Omron Sysmac Studio project SorterKonveyor (Sysmac Studio 1.65.0.64007, StandardProject)

# Controller new_Controller_0: NX1P2-1040DT1 version 1.69
Task PrimaryTask (priority 4, period or condition 2000): Program0

VAR_GLOBAL
    BIO_Input_Bit_00 : BOOL;  (* at BuiltInIO://cpu/#0/Input_Bit_00 *)
    BIO_Input_Bit_01 : BOOL;  (* at BuiltInIO://cpu/#0/Input_Bit_01 *)
    BIO_Input_Bit_02 : BOOL;  (* at BuiltInIO://cpu/#0/Input_Bit_02 *)
    BIO_Input_Bit_03 : BOOL;  (* at BuiltInIO://cpu/#0/Input_Bit_03 *)
    BIO_Input_Bit_04 : BOOL;  (* at BuiltInIO://cpu/#0/Input_Bit_04 *)
    BIO_Input_Bit_05 : BOOL;  (* at BuiltInIO://cpu/#0/Input_Bit_05 *)
    BIO_Input_Bit_06 : BOOL;  (* at BuiltInIO://cpu/#0/Input_Bit_06 *)
    BIO_Input_Bit_07 : BOOL;  (* at BuiltInIO://cpu/#0/Input_Bit_07 *)
    BIO_Output_Bit_00 : BOOL;  (* at BuiltInIO://cpu/#0/Output_Bit_00 *)
    BIO_Output_Bit_01 : BOOL;  (* at BuiltInIO://cpu/#0/Output_Bit_01 *)
    BIO_Output_Bit_02 : BOOL;  (* at BuiltInIO://cpu/#0/Output_Bit_02 *)
    BIO_Output_Bit_03 : BOOL;  (* at BuiltInIO://cpu/#0/Output_Bit_03 *)
    BIO_Output_Bit_04 : BOOL;  (* at BuiltInIO://cpu/#0/Output_Bit_04 *)
    BIO_Output_Bit_05 : BOOL;  (* at BuiltInIO://cpu/#0/Output_Bit_05 *)
    BIO_Output_Bit_06 : BOOL;  (* at BuiltInIO://cpu/#0/Output_Bit_06 *)
    BIO_Output_Bit_07 : BOOL;  (* at BuiltInIO://cpu/#0/Output_Bit_07 *)
    BIO_Output_Bit_08 : BOOL;  (* at BuiltInIO://cpu/#0/Output_Bit_08 *)
    BIO_Output_Bit_09 : BOOL;  (* at BuiltInIO://cpu/#0/Output_Bit_09 *)
    IN_Start_But : BOOL;
    IN_Stop_But : BOOL;
    IN_Motor0_Ariza : BOOL;
    IN_Motor1_Ariza : BOOL;
    IN_Motor3_Ariza : BOOL;
    IN_Motor2_Ariza : BOOL;
    IN_Motor4_Ariza : BOOL;
    OUT_Motor0_İleri : BOOL;
    OUT_Motor0_Geri : BOOL;
    OUT_Motor1_İleri : BOOL;
    OUT_Motor1_Geri : BOOL;
    OUT_Motor2_İleri : BOOL;
    OUT_Motor2_Geri : BOOL;
    OUT_Motor3_İleri : BOOL;
    OUT_Motor3_Geri : BOOL;
    OUT_Motor4_İleri : BOOL;
    OUT_Motor4_Geri : BOOL;
    OUT_Buzzer : BOOL;
    IN_Urun_Algilama_Sens : BOOL;
    ALARM : ARRAY[0..50] OF BOOL;
    Barcode_Info : STRING[10];
    Product_Cycle : INT;
    Barcode_Regsiter1 : STRING[10];
    Barcode_Regsiter2 : STRING[10];
    Barcode_Regsiter3 : STRING[10];
    Barcode_Regsiter4 : STRING[10];
    Barcode_Regsiter5 : STRING[10];
    Barcode_Regsiter6 : STRING[10];
    Barcode_Regsiter7 : STRING[10];
    Barcode_Regsiter8 : STRING[10];
    Barcode_Regsiter9 : STRING[10];
    Barcode_Regsiter10 : STRING[10];
    PC1_Reset : BOOL;
    PC2_Reset : BOOL;
    PC3_Reset : BOOL;
    PC4_Reset : BOOL;
    PC5_Reset : BOOL;
    PC6_Reset : BOOL;
    PC8_Reset : BOOL;
    PC7_Reset : BOOL;
    PC9_Reset : BOOL;
    PC10_Reset : BOOL;
    Urun_Eslesmedi_Alarmi : BOOL;
END_VAR

PROGRAM Program0
VAR
    Buzzer : BOOL;
    TON_Buzzer : TON;
    Safety_OK : BOOL;
    syc : INT;
    PC1 : BOOL;
    PC2 : BOOL;
    PC3 : BOOL;
    PC4 : BOOL;
    PC5 : BOOL;
    PC6 : BOOL;
    PC7 : BOOL;
    PC8 : BOOL;
    PC9 : BOOL;
    PC10 : BOOL;
    PC1_AllTime : AccumulationTimer;
    PC2_AllTime : AccumulationTimer;
    PC10_AllTime : AccumulationTimer;
    PC9_AllTime : AccumulationTimer;
    PC8_AllTime : AccumulationTimer;
    PC7_AllTime : AccumulationTimer;
    PC6_AllTime : AccumulationTimer;
    PC5_AllTime : AccumulationTimer;
    PC4_AllTime : AccumulationTimer;
    PC3_AllTime : AccumulationTimer;
    TOF1_Calisma : TOF;
    TOF2_Calisma : TOF;
    TOF3_Calisma : TOF;
    TOF4_Calisma : TOF;
    TOF5_Calisma : TOF;
END_VAR
VAR_EXTERNAL
    BIO_Input_Bit_00 : BOOL;
    BIO_Input_Bit_01 : BOOL;
    BIO_Input_Bit_02 : BOOL;
    BIO_Input_Bit_03 : BOOL;
    BIO_Input_Bit_04 : BOOL;
    BIO_Input_Bit_05 : BOOL;
    IN_Start_But : BOOL;
    IN_Stop_But : BOOL;
    IN_Motor0_Ariza : BOOL;
    IN_Motor1_Ariza : BOOL;
    IN_Motor3_Ariza : BOOL;
    IN_Motor2_Ariza : BOOL;
    BIO_Input_Bit_06 : BOOL;
    IN_Motor4_Ariza : BOOL;
    BIO_Output_Bit_00 : BOOL;
    BIO_Output_Bit_01 : BOOL;
    BIO_Output_Bit_02 : BOOL;
    BIO_Output_Bit_03 : BOOL;
    BIO_Output_Bit_04 : BOOL;
    BIO_Output_Bit_05 : BOOL;
    BIO_Output_Bit_06 : BOOL;
    BIO_Output_Bit_07 : BOOL;
    BIO_Output_Bit_08 : BOOL;
    OUT_Motor0_İleri : BOOL;
    OUT_Motor0_Geri : BOOL;
    OUT_Motor1_İleri : BOOL;
    OUT_Motor1_Geri : BOOL;
    OUT_Motor2_İleri : BOOL;
    OUT_Motor2_Geri : BOOL;
    OUT_Motor3_İleri : BOOL;
    OUT_Motor3_Geri : BOOL;
    OUT_Motor4_İleri : BOOL;
    OUT_Motor4_Geri : BOOL;
    OUT_Buzzer : BOOL;
    BIO_Output_Bit_09 : BOOL;
    BIO_Input_Bit_07 : BOOL;
    IN_Urun_Algilama_Sens : BOOL;
    ALARM : ARRAY[0..50] OF BOOL;
    Barcode_Info : STRING[10];
    Product_Cycle : INT;
    Barcode_Regsiter1 : STRING[10];
    Barcode_Regsiter2 : STRING[10];
    Barcode_Regsiter3 : STRING[10];
    Barcode_Regsiter4 : STRING[10];
    Barcode_Regsiter5 : STRING[10];
    Barcode_Regsiter6 : STRING[10];
    Barcode_Regsiter7 : STRING[10];
    Barcode_Regsiter8 : STRING[10];
    Barcode_Regsiter9 : STRING[10];
    Barcode_Regsiter10 : STRING[10];
    PC1_Reset : BOOL;
    PC2_Reset : BOOL;
    PC3_Reset : BOOL;
    PC4_Reset : BOOL;
    PC5_Reset : BOOL;
    PC6_Reset : BOOL;
    PC8_Reset : BOOL;
    PC7_Reset : BOOL;
    PC9_Reset : BOOL;
    PC10_Reset : BOOL;
    Urun_Eslesmedi_Alarmi : BOOL;
END_VAR
VAR
    _e1 : R_TRIG;
    _e2 : R_TRIG;
    _e3 : R_TRIG;
    _e4 : R_TRIG;
    _e5 : R_TRIG;
    _e6 : R_TRIG;
    _e7 : R_TRIG;
    _e8 : R_TRIG;
    _e9 : R_TRIG;
    _e10 : R_TRIG;
    _e11 : R_TRIG;
    _e12 : R_TRIG;
    _e13 : R_TRIG;
    _e14 : R_TRIG;
    _e15 : R_TRIG;
    _e16 : R_TRIG;
    _e17 : R_TRIG;
    _e18 : R_TRIG;
    _e19 : R_TRIG;
    _e20 : R_TRIG;
    _e21 : R_TRIG;
    _e22 : R_TRIG;
    _e23 : R_TRIG;
END_VAR

(* Section InOut: ladder, written here as Structured Text *)

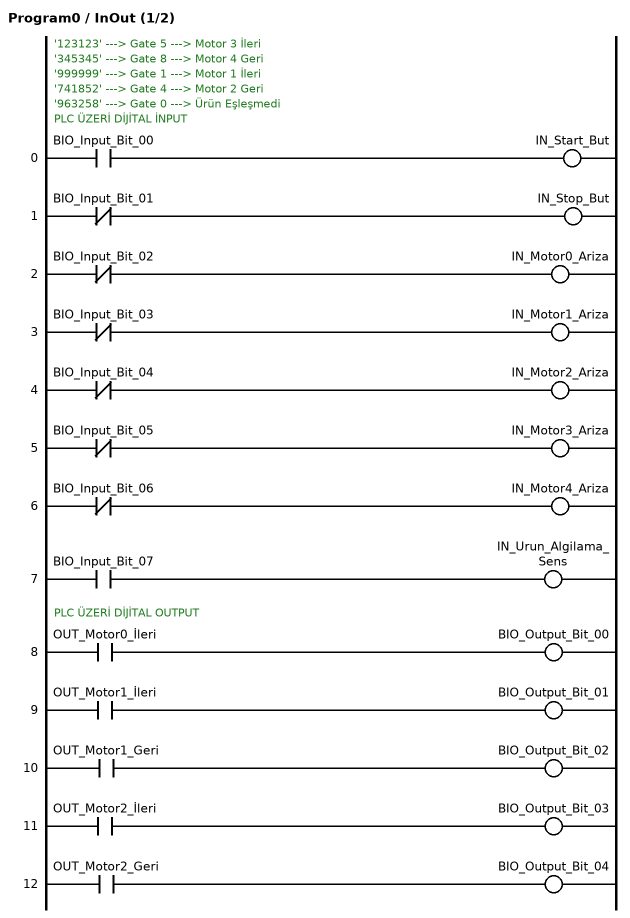
(* Rung 0: '123123' ---> Gate 5 ---> Motor 3 İleri / '345345' ---> Gate 8 ---> Motor 4 Geri / '999999' ---> Gate 1 ---> Motor 1 İleri / '741852' ---> Gate 4 ---> Motor 2 Geri / '963258' ---> Gate 0 ---> Ürün Eşleşmedi / PLC ÜZERİ DİJİTAL İNPUT *)
IN_Start_But := BIO_Input_Bit_00;
(* Rung 1 *)
IN_Stop_But := NOT BIO_Input_Bit_01;
(* Rung 2 *)
IN_Motor0_Ariza := NOT BIO_Input_Bit_02;
(* Rung 3 *)
IN_Motor1_Ariza := NOT BIO_Input_Bit_03;
(* Rung 4 *)
IN_Motor2_Ariza := NOT BIO_Input_Bit_04;
(* Rung 5 *)
IN_Motor3_Ariza := NOT BIO_Input_Bit_05;
(* Rung 6 *)
IN_Motor4_Ariza := NOT BIO_Input_Bit_06;
(* Rung 7 *)
IN_Urun_Algilama_Sens := BIO_Input_Bit_07;
(* Rung 8: PLC ÜZERİ DİJİTAL OUTPUT *)
BIO_Output_Bit_00 := OUT_Motor0_İleri;
(* Rung 9 *)
BIO_Output_Bit_01 := OUT_Motor1_İleri;
(* Rung 10 *)
BIO_Output_Bit_02 := OUT_Motor1_Geri;
(* Rung 11 *)
BIO_Output_Bit_03 := OUT_Motor2_İleri;
(* Rung 12 *)
BIO_Output_Bit_04 := OUT_Motor2_Geri;

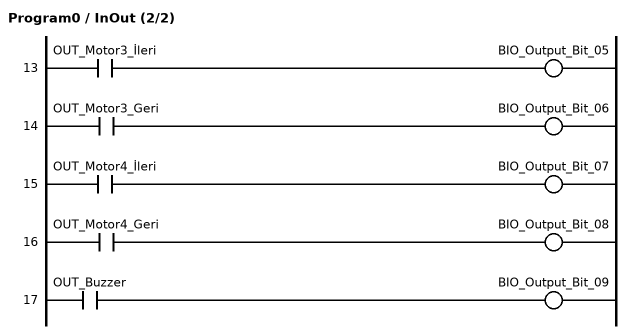
(* Rung 13 *)
BIO_Output_Bit_05 := OUT_Motor3_İleri;
(* Rung 14 *)
BIO_Output_Bit_06 := OUT_Motor3_Geri;
(* Rung 15 *)
BIO_Output_Bit_07 := OUT_Motor4_İleri;
(* Rung 16 *)
BIO_Output_Bit_08 := OUT_Motor4_Geri;
(* Rung 17 *)
BIO_Output_Bit_09 := OUT_Buzzer;

(* Section Alarmlar: ladder, written here as Structured Text *)

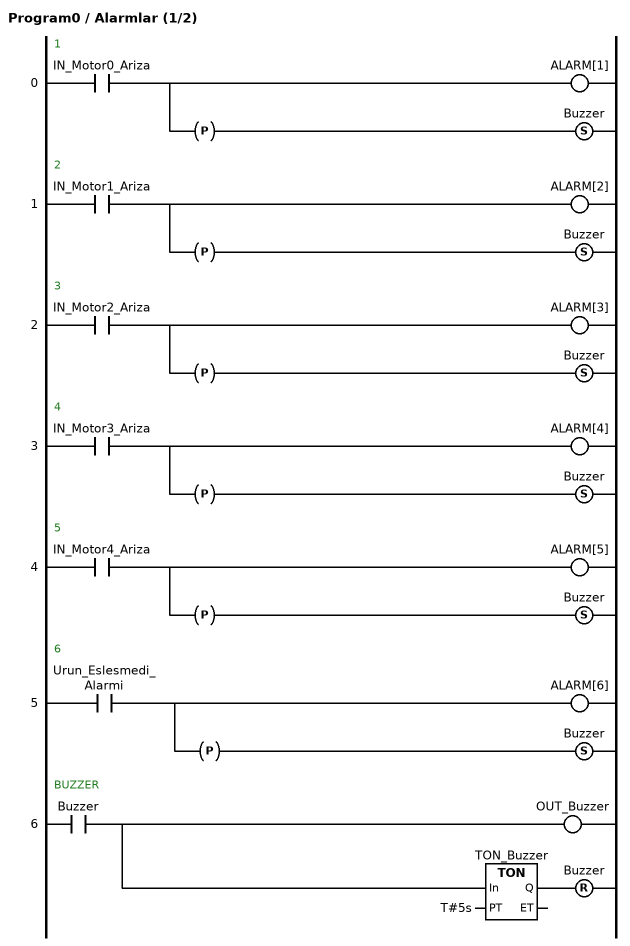
(* Rung 0: 1 *)
ALARM[1] := IN_Motor0_Ariza;
_e1(CLK := IN_Motor0_Ariza);
IF _e1.Q THEN Buzzer := TRUE; END_IF;
(* Rung 1: 2 *)
ALARM[2] := IN_Motor1_Ariza;
_e2(CLK := IN_Motor1_Ariza);
IF _e2.Q THEN Buzzer := TRUE; END_IF;
(* Rung 2: 3 *)
ALARM[3] := IN_Motor2_Ariza;
_e3(CLK := IN_Motor2_Ariza);
IF _e3.Q THEN Buzzer := TRUE; END_IF;
(* Rung 3: 4 *)
ALARM[4] := IN_Motor3_Ariza;
_e4(CLK := IN_Motor3_Ariza);
IF _e4.Q THEN Buzzer := TRUE; END_IF;
(* Rung 4: 5 *)
ALARM[5] := IN_Motor4_Ariza;
_e5(CLK := IN_Motor4_Ariza);
IF _e5.Q THEN Buzzer := TRUE; END_IF;
(* Rung 5: 6 *)
ALARM[6] := Urun_Eslesmedi_Alarmi;
_e6(CLK := Urun_Eslesmedi_Alarmi);
IF _e6.Q THEN Buzzer := TRUE; END_IF;
(* Rung 6: BUZZER *)
OUT_Buzzer := Buzzer;
TON_Buzzer(In := Buzzer, PT := T#5s);
IF TON_Buzzer.Q THEN Buzzer := FALSE; END_IF;

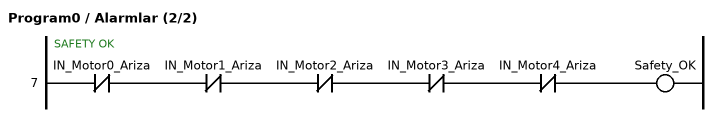
(* Rung 7: SAFETY OK *)
Safety_OK := NOT IN_Motor0_Ariza AND NOT IN_Motor1_Ariza AND NOT IN_Motor2_Ariza AND NOT IN_Motor3_Ariza AND NOT IN_Motor4_Ariza;

(* Section Urun_Tasima: ladder, written here as Structured Text *)

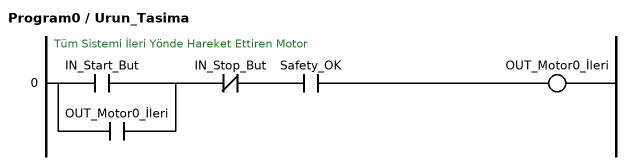
(* Rung 0: Tüm Sistemi İleri Yönde Hareket Ettiren Motor *)
OUT_Motor0_İleri := (IN_Start_But OR OUT_Motor0_İleri) AND NOT IN_Stop_But AND Safety_OK;

(* Section Barkoddan_Bilgi_Man: ladder, written here as Structured Text *)

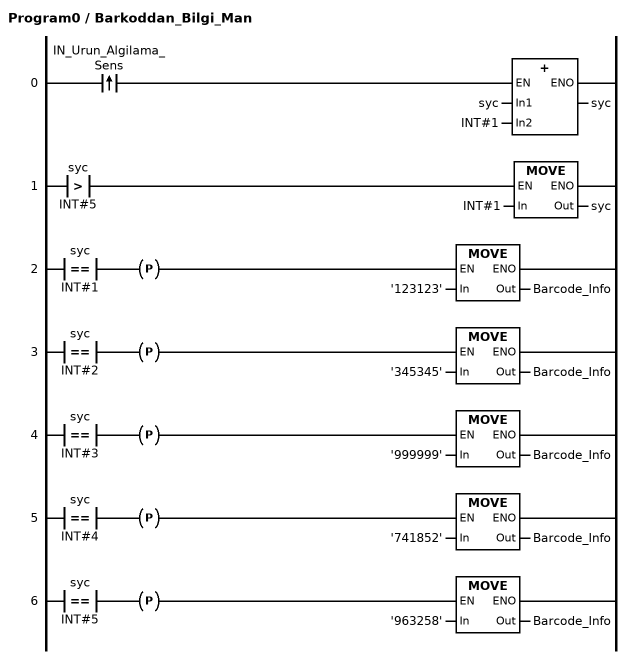
(* Rung 0 *)
_e7(CLK := IN_Urun_Algilama_Sens);
IF _e7.Q THEN syc := syc + INT#1; END_IF;
(* Rung 1 *)
IF syc > INT#5 THEN syc := INT#1; END_IF;
(* Rung 2 *)
_e8(CLK := syc = INT#1);
IF _e8.Q THEN Barcode_Info := '123123'; END_IF;
(* Rung 3 *)
_e9(CLK := syc = INT#2);
IF _e9.Q THEN Barcode_Info := '345345'; END_IF;
(* Rung 4 *)
_e10(CLK := syc = INT#3);
IF _e10.Q THEN Barcode_Info := '999999'; END_IF;
(* Rung 5 *)
_e11(CLK := syc = INT#4);
IF _e11.Q THEN Barcode_Info := '741852'; END_IF;
(* Rung 6 *)
_e12(CLK := syc = INT#5);
IF _e12.Q THEN Barcode_Info := '963258'; END_IF;

(* Section Buffer: ladder, written here as Structured Text *)

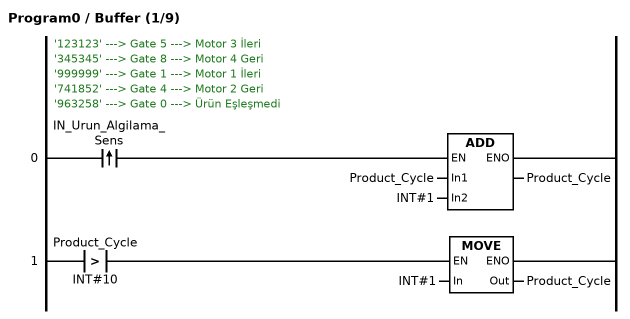
(* Rung 0: '123123' ---> Gate 5 ---> Motor 3 İleri / '345345' ---> Gate 8 ---> Motor 4 Geri / '999999' ---> Gate 1 ---> Motor 1 İleri / '741852' ---> Gate 4 ---> Motor 2 Geri / '963258' ---> Gate 0 ---> Ürün Eşleşmedi *)
_e13(CLK := IN_Urun_Algilama_Sens);
IF _e13.Q THEN Product_Cycle := Product_Cycle + INT#1; END_IF;
(* Rung 1 *)
IF Product_Cycle > INT#10 THEN Product_Cycle := INT#1; END_IF;

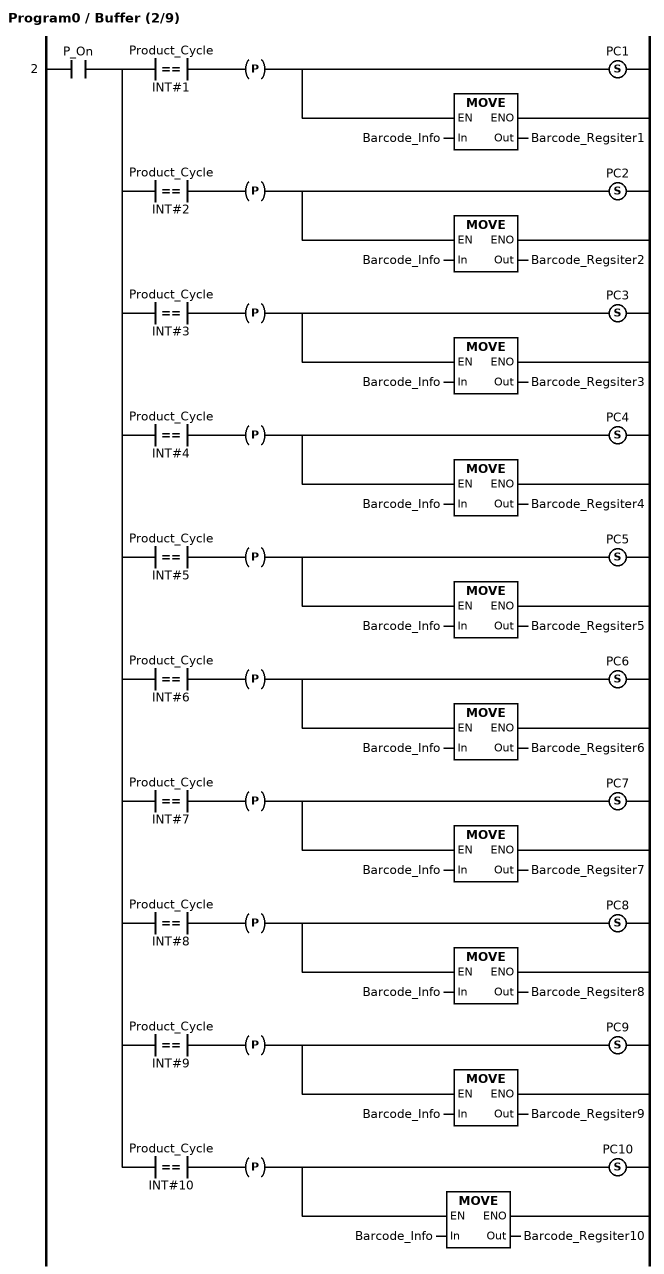
(* Rung 2 *)
_e14(CLK := P_On AND (Product_Cycle = INT#1));
IF _e14.Q THEN
    PC1 := TRUE;
    Barcode_Regsiter1 := Barcode_Info;
END_IF;
_e15(CLK := P_On AND (Product_Cycle = INT#2));
IF _e15.Q THEN
    PC2 := TRUE;
    Barcode_Regsiter2 := Barcode_Info;
END_IF;
_e16(CLK := P_On AND (Product_Cycle = INT#3));
IF _e16.Q THEN
    PC3 := TRUE;
    Barcode_Regsiter3 := Barcode_Info;
END_IF;
_e17(CLK := P_On AND (Product_Cycle = INT#4));
IF _e17.Q THEN
    PC4 := TRUE;
    Barcode_Regsiter4 := Barcode_Info;
END_IF;
_e18(CLK := P_On AND (Product_Cycle = INT#5));
IF _e18.Q THEN
    PC5 := TRUE;
    Barcode_Regsiter5 := Barcode_Info;
END_IF;
_e19(CLK := P_On AND (Product_Cycle = INT#6));
IF _e19.Q THEN
    PC6 := TRUE;
    Barcode_Regsiter6 := Barcode_Info;
END_IF;
_e20(CLK := P_On AND (Product_Cycle = INT#7));
IF _e20.Q THEN
    PC7 := TRUE;
    Barcode_Regsiter7 := Barcode_Info;
END_IF;
_e21(CLK := P_On AND (Product_Cycle = INT#8));
IF _e21.Q THEN
    PC8 := TRUE;
    Barcode_Regsiter8 := Barcode_Info;
END_IF;
_e22(CLK := P_On AND (Product_Cycle = INT#9));
IF _e22.Q THEN
    PC9 := TRUE;
    Barcode_Regsiter9 := Barcode_Info;
END_IF;
_e23(CLK := P_On AND (Product_Cycle = INT#10));
IF _e23.Q THEN
    PC10 := TRUE;
    Barcode_Regsiter10 := Barcode_Info;
END_IF;

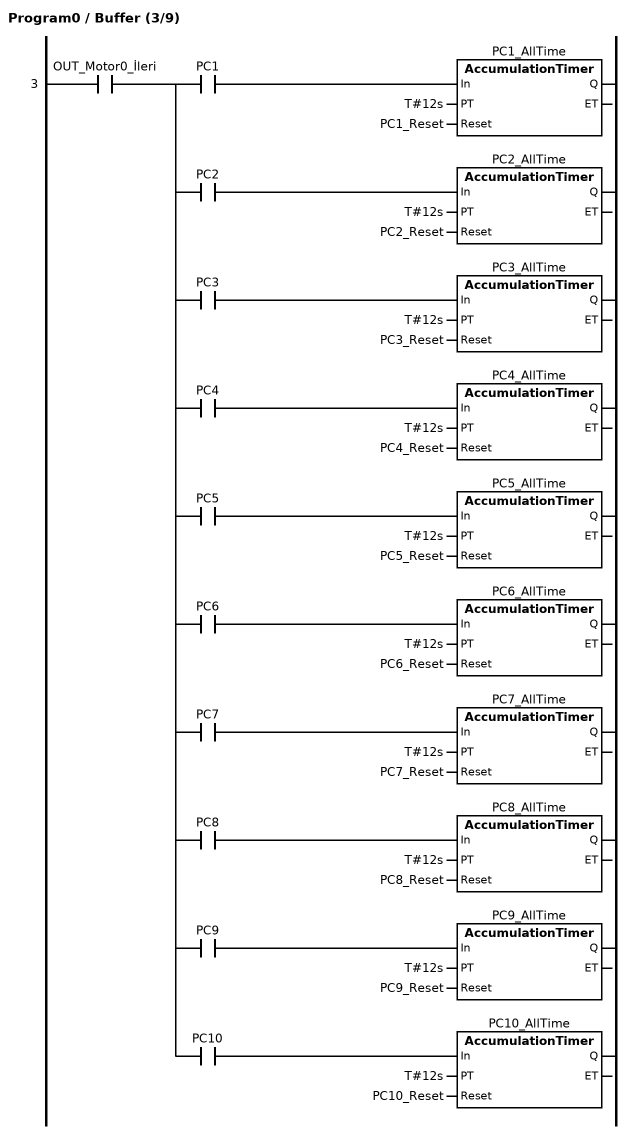
(* Rung 3 *)
PC1_AllTime(In := OUT_Motor0_İleri AND PC1, PT := T#12s, Reset := PC1_Reset);
PC2_AllTime(In := OUT_Motor0_İleri AND PC2, PT := T#12s, Reset := PC2_Reset);
PC3_AllTime(In := OUT_Motor0_İleri AND PC3, PT := T#12s, Reset := PC3_Reset);
PC4_AllTime(In := OUT_Motor0_İleri AND PC4, PT := T#12s, Reset := PC4_Reset);
PC5_AllTime(In := OUT_Motor0_İleri AND PC5, PT := T#12s, Reset := PC5_Reset);
PC6_AllTime(In := OUT_Motor0_İleri AND PC6, PT := T#12s, Reset := PC6_Reset);
PC7_AllTime(In := OUT_Motor0_İleri AND PC7, PT := T#12s, Reset := PC7_Reset);
PC8_AllTime(In := OUT_Motor0_İleri AND PC8, PT := T#12s, Reset := PC8_Reset);
PC9_AllTime(In := OUT_Motor0_İleri AND PC9, PT := T#12s, Reset := PC9_Reset);
PC10_AllTime(In := OUT_Motor0_İleri AND PC10, PT := T#12s, Reset := PC10_Reset);

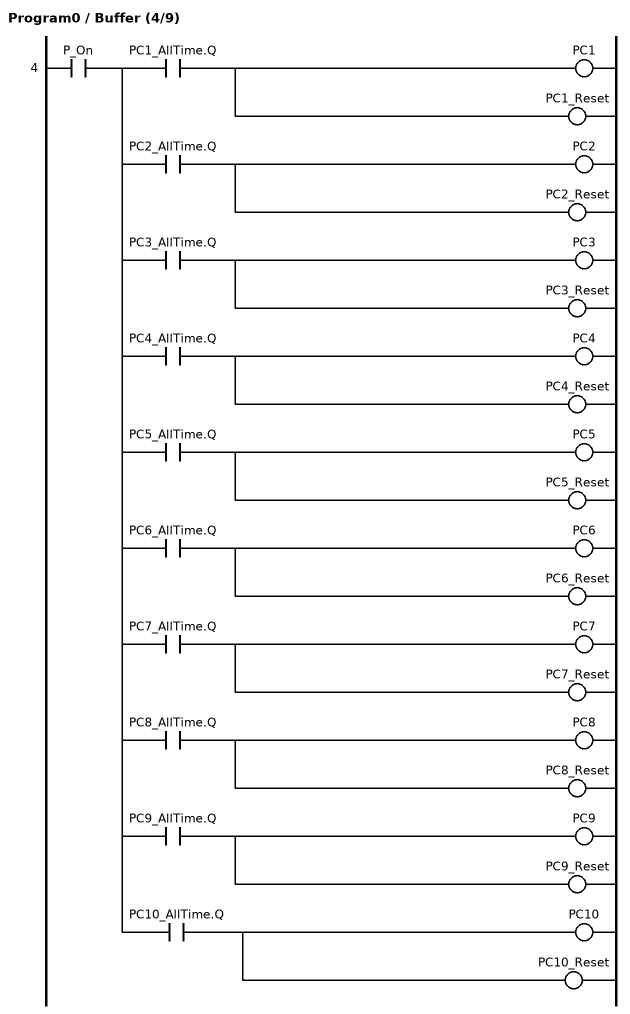
(* Rung 4 *)
PC1 := P_On AND PC1_AllTime.Q;
PC1_Reset := P_On AND PC1_AllTime.Q;
PC2 := P_On AND PC2_AllTime.Q;
PC2_Reset := P_On AND PC2_AllTime.Q;
PC3 := P_On AND PC3_AllTime.Q;
PC3_Reset := P_On AND PC3_AllTime.Q;
PC4 := P_On AND PC4_AllTime.Q;
PC4_Reset := P_On AND PC4_AllTime.Q;
PC5 := P_On AND PC5_AllTime.Q;
PC5_Reset := P_On AND PC5_AllTime.Q;
PC6 := P_On AND PC6_AllTime.Q;
PC6_Reset := P_On AND PC6_AllTime.Q;
PC7 := P_On AND PC7_AllTime.Q;
PC7_Reset := P_On AND PC7_AllTime.Q;
PC8 := P_On AND PC8_AllTime.Q;
PC8_Reset := P_On AND PC8_AllTime.Q;
PC9 := P_On AND PC9_AllTime.Q;
PC9_Reset := P_On AND PC9_AllTime.Q;
PC10 := P_On AND PC10_AllTime.Q;
PC10_Reset := P_On AND PC10_AllTime.Q;

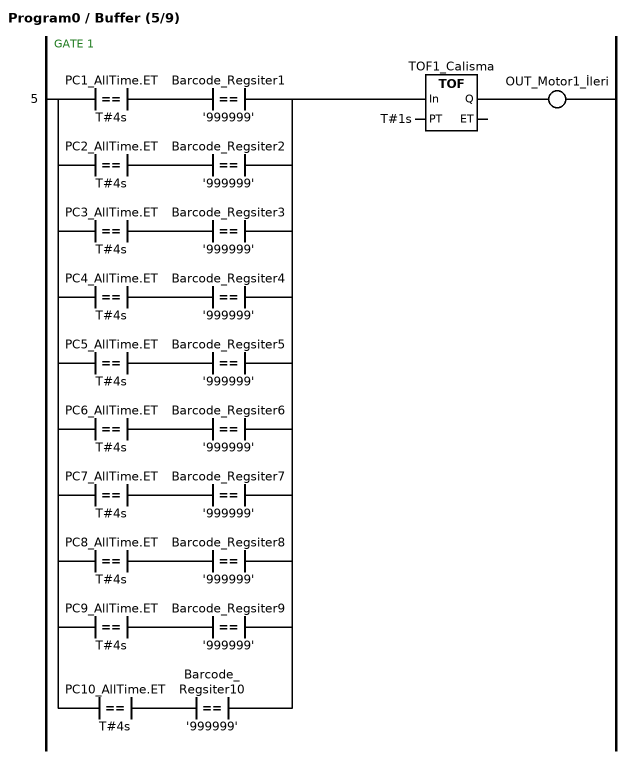
(* Rung 5: GATE 1 *)
TOF1_Calisma(In := ((PC1_AllTime.ET = T#4s) AND (Barcode_Regsiter1 = '999999')) OR ((PC2_AllTime.ET = T#4s) AND (Barcode_Regsiter2 = '999999')) OR ((PC3_AllTime.ET = T#4s) AND (Barcode_Regsiter3 = '999999')) OR ((PC4_AllTime.ET = T#4s) AND (Barcode_Regsiter4 = '999999')) OR ((PC5_AllTime.ET = T#4s) AND (Barcode_Regsiter5 = '999999')) OR ((PC6_AllTime.ET = T#4s) AND (Barcode_Regsiter6 = '999999')) OR ((PC7_AllTime.ET = T#4s) AND (Barcode_Regsiter7 = '999999')) OR ((PC8_AllTime.ET = T#4s) AND (Barcode_Regsiter8 = '999999')) OR ((PC9_AllTime.ET = T#4s) AND (Barcode_Regsiter9 = '999999')) OR ((PC10_AllTime.ET = T#4s) AND (Barcode_Regsiter10 = '999999')), PT := T#1s);
OUT_Motor1_İleri := TOF1_Calisma.Q;

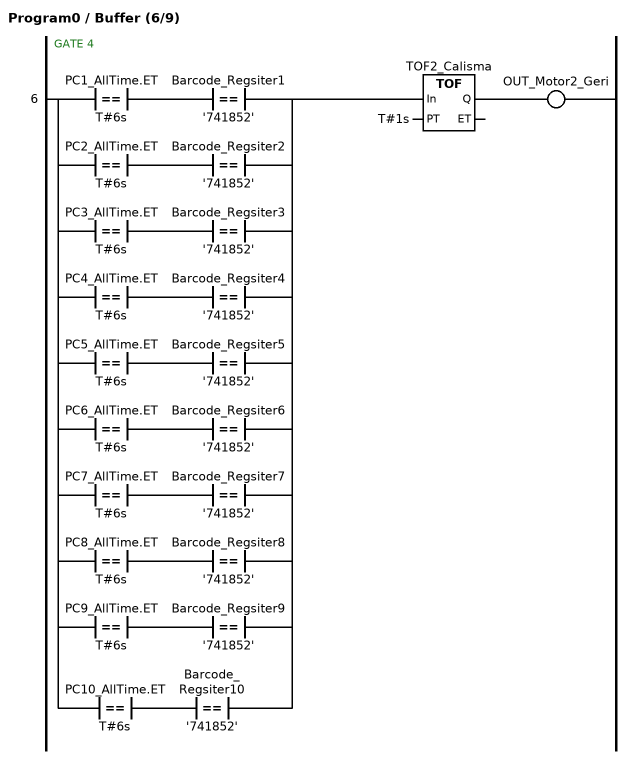
(* Rung 6: GATE 4 *)
TOF2_Calisma(In := ((PC1_AllTime.ET = T#6s) AND (Barcode_Regsiter1 = '741852')) OR ((PC2_AllTime.ET = T#6s) AND (Barcode_Regsiter2 = '741852')) OR ((PC3_AllTime.ET = T#6s) AND (Barcode_Regsiter3 = '741852')) OR ((PC4_AllTime.ET = T#6s) AND (Barcode_Regsiter4 = '741852')) OR ((PC5_AllTime.ET = T#6s) AND (Barcode_Regsiter5 = '741852')) OR ((PC6_AllTime.ET = T#6s) AND (Barcode_Regsiter6 = '741852')) OR ((PC7_AllTime.ET = T#6s) AND (Barcode_Regsiter7 = '741852')) OR ((PC8_AllTime.ET = T#6s) AND (Barcode_Regsiter8 = '741852')) OR ((PC9_AllTime.ET = T#6s) AND (Barcode_Regsiter9 = '741852')) OR ((PC10_AllTime.ET = T#6s) AND (Barcode_Regsiter10 = '741852')), PT := T#1s);
OUT_Motor2_Geri := TOF2_Calisma.Q;

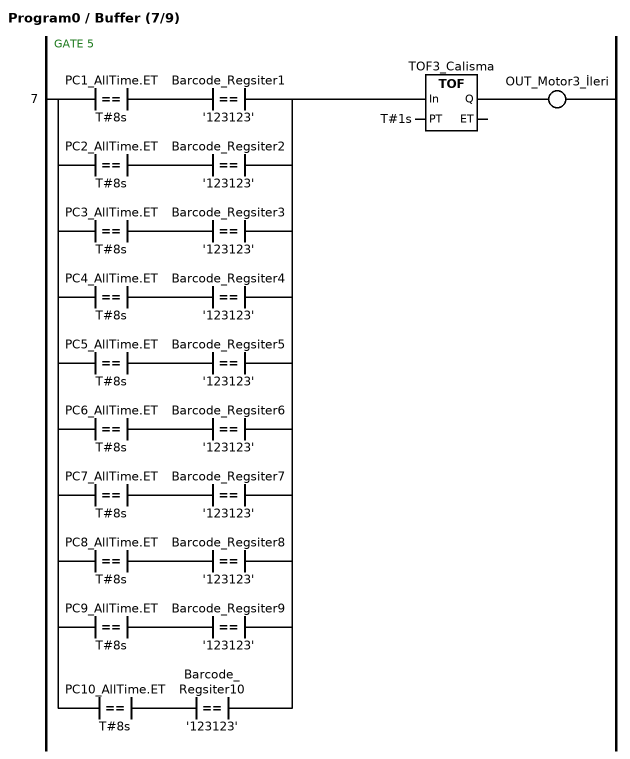
(* Rung 7: GATE 5 *)
TOF3_Calisma(In := ((PC1_AllTime.ET = T#8s) AND (Barcode_Regsiter1 = '123123')) OR ((PC2_AllTime.ET = T#8s) AND (Barcode_Regsiter2 = '123123')) OR ((PC3_AllTime.ET = T#8s) AND (Barcode_Regsiter3 = '123123')) OR ((PC4_AllTime.ET = T#8s) AND (Barcode_Regsiter4 = '123123')) OR ((PC5_AllTime.ET = T#8s) AND (Barcode_Regsiter5 = '123123')) OR ((PC6_AllTime.ET = T#8s) AND (Barcode_Regsiter6 = '123123')) OR ((PC7_AllTime.ET = T#8s) AND (Barcode_Regsiter7 = '123123')) OR ((PC8_AllTime.ET = T#8s) AND (Barcode_Regsiter8 = '123123')) OR ((PC9_AllTime.ET = T#8s) AND (Barcode_Regsiter9 = '123123')) OR ((PC10_AllTime.ET = T#8s) AND (Barcode_Regsiter10 = '123123')), PT := T#1s);
OUT_Motor3_İleri := TOF3_Calisma.Q;

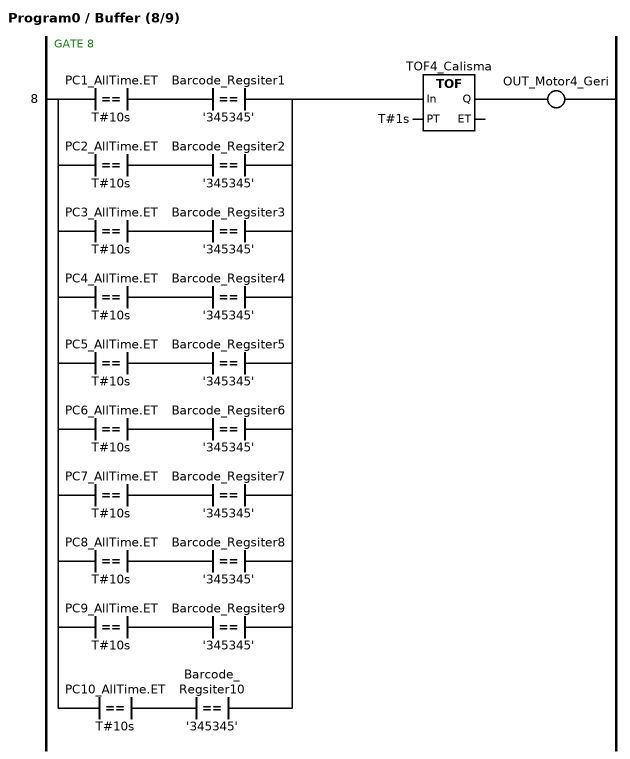
(* Rung 8: GATE 8 *)
TOF4_Calisma(In := ((PC1_AllTime.ET = T#10s) AND (Barcode_Regsiter1 = '345345')) OR ((PC2_AllTime.ET = T#10s) AND (Barcode_Regsiter2 = '345345')) OR ((PC3_AllTime.ET = T#10s) AND (Barcode_Regsiter3 = '345345')) OR ((PC4_AllTime.ET = T#10s) AND (Barcode_Regsiter4 = '345345')) OR ((PC5_AllTime.ET = T#10s) AND (Barcode_Regsiter5 = '345345')) OR ((PC6_AllTime.ET = T#10s) AND (Barcode_Regsiter6 = '345345')) OR ((PC7_AllTime.ET = T#10s) AND (Barcode_Regsiter7 = '345345')) OR ((PC8_AllTime.ET = T#10s) AND (Barcode_Regsiter8 = '345345')) OR ((PC9_AllTime.ET = T#10s) AND (Barcode_Regsiter9 = '345345')) OR ((PC10_AllTime.ET = T#10s) AND (Barcode_Regsiter10 = '345345')), PT := T#1s);
OUT_Motor4_Geri := TOF4_Calisma.Q;

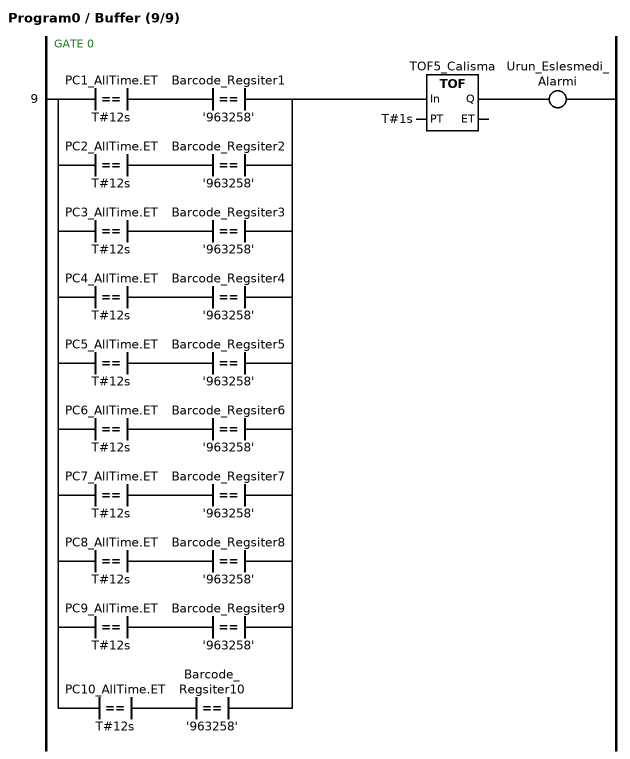
(* Rung 9: GATE 0 *)
TOF5_Calisma(In := ((PC1_AllTime.ET = T#12s) AND (Barcode_Regsiter1 = '963258')) OR ((PC2_AllTime.ET = T#12s) AND (Barcode_Regsiter2 = '963258')) OR ((PC3_AllTime.ET = T#12s) AND (Barcode_Regsiter3 = '963258')) OR ((PC4_AllTime.ET = T#12s) AND (Barcode_Regsiter4 = '963258')) OR ((PC5_AllTime.ET = T#12s) AND (Barcode_Regsiter5 = '963258')) OR ((PC6_AllTime.ET = T#12s) AND (Barcode_Regsiter6 = '963258')) OR ((PC7_AllTime.ET = T#12s) AND (Barcode_Regsiter7 = '963258')) OR ((PC8_AllTime.ET = T#12s) AND (Barcode_Regsiter8 = '963258')) OR ((PC9_AllTime.ET = T#12s) AND (Barcode_Regsiter9 = '963258')) OR ((PC10_AllTime.ET = T#12s) AND (Barcode_Regsiter10 = '963258')), PT := T#1s);
Urun_Eslesmedi_Alarmi := TOF5_Calisma.Q;
END_PROGRAM